// TIA Portal V21 export
FUNCTION "Scala" : Void   // FC2191, LAD
{ S7_Optimized_Access := 'TRUE' }
// stored: IsIECCheckEnabled true, SetENOAutomatically false
   VAR_INPUT
      ValoreIn : Real;
      MaxLimitInput : Real;
      MinLimitInput : Real;
      MaxLimitOut : Real;
      MinLimitOut : Real;
   END_VAR
   VAR_IN_OUT
      ValoreOut : Real;
   END_VAR
   VAR_TEMP
      AnologInput : Real;
      Output_Range : Real;
      Input_Range : Real;
      Kangolare : Real;
   END_VAR
BEGIN

REGION Network 1 (SCL)
   REGION Ingressi
       #AnologInput := #ValoreIn;
   END_REGION ;
   REGION limiti ingresso
       IF #AnologInput > #MaxLimitInput THEN
           #AnologInput := #MaxLimitInput;
       END_IF;
   END_REGION ;
   REGION Calcolo
       #Output_Range := #MaxLimitOut - #MinLimitOut;
       #Input_Range := #MaxLimitInput - #MinLimitInput;
       #Kangolare := #Output_Range / #Input_Range;

       #ValoreOut := ((#AnologInput - #MaxLimitInput) * #Kangolare) + #MaxLimitOut;
   END_REGION ;
   REGION limiti uscita
       IF #ValoreOut > #MaxLimitOut THEN
           #ValoreOut := #MaxLimitOut;
       END_IF;
       IF #ValoreOut < #MinLimitOut THEN
           #ValoreOut := #MinLimitOut;
       END_IF;
   END_REGION ;
END_REGION
END_FUNCTION
